FUNCTION_BLOCK FB_MotorControlReverse EXTENDS FB_MotorControl
VAR
	reverseButton		: Button;	// Scada Button reverse
	iDriveReverse		: I_DriveReverse; //Interface variable 
	
	bSuccess: BOOL;
	
END_VAR

SUPER^(); //call base class 

//Button Auto is set in SCADA motor control station, but Client in PLC have to have acces too directly via a variable to work in Auto mode
IF autoButton.IsPressed THEN 
	AutoOn();	// Turn On SCADA auto Led
ELSE
	AutoOff(); // Turn Off SCADA auto Led
	
	// IF NOT AUTO MODE THEN, EXECUTE
	
	CASE eStateDevice OF
		eOn :
			 IF reverseButton.IsPressed THEN
				ReverseOn();
			 END_IF
				 
		eOff :
			ReverseOff();
			iDrive.WorkCounterOff();
				
		eReverse :
			IF reverseButton.IsPressed THEN
            	iDrive.WorkCount();			
				iDrive.WorkCounterOn();
			ELSE	
				ReverseOff();
				iDrive.WorkCounterOff();
			 END_IF
		
		eFault :
			ReverseOff();
			iDrive.WorkCounterOff();
	
	END_CASE

END_IF

METHOD FB_init : BOOL
VAR_INPUT
	bInitRetains : BOOL; // if TRUE, the retain variables are initialized (warm start / cold start)
	bInCopyCode  : BOOL;  // if TRUE, the instance afterwards gets moved into the copy code (online change)
	iDrive		 : I_Drive;
			
END_VAR
//check it is possible conversion type of interface

IF __QUERYINTERFACE(iDrive, iDriveReverse) THEN
	bSuccess := TRUE;
END_IF
END_METHOD

METHOD ReverseOff : BOOL
VAR_INPUT
END_VAR
iDriveReverse.SwitchReverseOff();
END_METHOD

METHOD ReverseOn : BOOL
VAR_INPUT
END_VAR
iDriveReverse.SwitchReverseOn();
END_METHOD

END_FUNCTION_BLOCK

(* stored: Version 1.1.0.1, ProductVersion 3.1.4024.12
   POU FB_MotorControlReverse: Id {e3f6163d-999c-4c4f-bc04-2ed30004ff70}, SpecialFunc None
   Method FB_init: Id {ae3fb759-2dd1-4395-b7cc-36f373dd76fb}
   Method ReverseOff: Id {755b010d-844a-4604-9bcb-4be64e1215bf}
   Method ReverseOn: Id {c76a633c-5fd6-4c8d-90e7-611a4362c596} *)
